{attribute 'GeneratedUsingTerminal: EP2316-0008-0018'}
{attribute addProperty BoxType "EP2316-0008-0018"}
{attribute addProperty Description "EP2316-0008 8 Ch. Dig. In, 10µs, 8Ch. Dig. Out 24V, 0,5A, Diagnostic, D-SUB25"}
{attribute addProperty Physics "YY"}
{attribute addProperty Id "DIG_InputsAT %I*DIG_Inputs_CC4551489DIG_Diag_InputsAT %I*DIG_Diag_Inputs_584303BF8DIG_Inputs_DeviceAT %I*DIG_Inputs_Device_4E5AF17E5DIG_OutputsAT %Q*DIG_Outputs_28AC1A9E8DIG_Outputs_DeviceAT %Q*DIG_Outputs_Device_36A5EF172WcStateAT %I*WcState_9091E0EB2InfoDataAT %I*InfoData_32EB74EA10"}
{attribute addProperty CRC "3704770447"}
{attribute addProperty Size "44"}
TYPE EP2316_DCD24F8F EXTENDS EtcSlaveBoxBase_77A0E4A7 :
STRUCT
	{attribute addProperty Name "DIG_Inputs"}
	DIG_Inputs : DIG_Inputs_CC455148;
	{attribute addProperty Name "DIG_Diag_Inputs"}
	DIG_Diag_Inputs : DIG_Diag_Inputs_584303BF;
	{attribute addProperty Name "DIG_Inputs_Device"}
	DIG_Inputs_Device : DIG_Inputs_Device_4E5AF17E;
	{attribute addProperty Name "DIG_Outputs"}
	DIG_Outputs : DIG_Outputs_28AC1A9E;
	{attribute addProperty Name "DIG_Outputs_Device"}
	DIG_Outputs_Device : DIG_Outputs_Device_36A5EF17;
	{attribute addProperty Name "WcState"}
	WcState : WcState_9091E0EB;
	{attribute addProperty Name "InfoData"}
	InfoData : InfoData_32EB74EA;
END_STRUCT
END_TYPE

(* stored: Version 1.2.0.0, ProductVersion 3.1.4024.9
   DUT EP2316_DCD24F8F: Id {48293bd9-5584-451e-9387-2a4806139019} *)
